FUNCTION_BLOCK GET_AT_INDEX (* Fetch value from array at given index. Array data type has to match with output data type. *)
  PACKAGE eclipse4diac::convert;
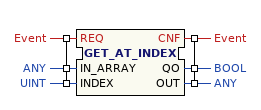
  EVENT_INPUT
    REQ WITH IN_ARRAY, INDEX; (* Service Request *)
  END_EVENT
  EVENT_OUTPUT
    CNF WITH QO, OUT; (* Confirmation of Requested Service *)
  END_EVENT
  VAR_INPUT
    IN_ARRAY : ANY; (* input array *)
    INDEX : UINT; (* index to fetch value from *)
  END_VAR
  VAR_OUTPUT
    QO : BOOL; (* Event Output Qualifier *)
    OUT : ANY; (* fetched output value *)
  END_VAR
END_FUNCTION_BLOCK
